{attribute 'GeneratedUsingTerminal: EL3612-0000-0016'}
{attribute addProperty BoxType "EL3612-0000-0016"}
{attribute addProperty Id "AI_Inputs_Channel_1AT %I*AI_Inputs_Channel_10B8F80A11AI_Inputs_Channel_2AT %I*AI_Inputs_Channel_10B8F80A11WcStateAT %I*WcState_9091E0EB2InfoDataAT %I*InfoData_94A18F5E2"}
{attribute addProperty CRC "1946162937"}
{attribute addProperty Size "26"}
TYPE EL3612_740016F9 EXTENDS EtcSlaveTerminalBase_947E5A46 :
STRUCT
	{attribute addProperty Name "AI_Inputs_Channel_1"}
	AI_Inputs_Channel_1 : AI_Inputs_Channel_10B8F80A;
	{attribute addProperty Name "AI_Inputs_Channel_2"}
	AI_Inputs_Channel_2 : AI_Inputs_Channel_10B8F80A;
	{attribute addProperty Name "WcState"}
	WcState : WcState_9091E0EB;
	{attribute addProperty Name "InfoData"}
	InfoData : InfoData_94A18F5E;
END_STRUCT
END_TYPE

(* stored: Version 1.2.0.0, ProductVersion 3.1.4024.9
   DUT EL3612_740016F9: Id {fb7cf138-12fd-422d-bc8b-2f3cac13c639} *)
